TYPE GVL_VLS :
STRUCT
END_STRUCT
END_TYPE

(* stored: Version 1.1.0.1, ProductVersion 3.1.4022.18
   DUT GVL_VLS: Id {c784d4bd-cd11-46ee-9046-ce523ddf74dd} *)
